TYPE ST_GAM_PIP :
STRUCT
	//Discrete Readback 
	xOn AT%I*:BOOL; //Readback of whether Gamma Ion Pump is turned on or not
END_STRUCT
END_TYPE

(* stored: Version 1.1.0.1, ProductVersion 3.1.4020.12
   DUT ST_GAM_PIP: Id {fa45bb55-ea5c-4be6-9451-79b23721a0cd} *)
